TYPE ST_LaudaReadCommands_Control :
STRUCT
	SetpointOffset	: STRING := 'IN_PAR_14_';
	ControlVariable	: STRING := 'IN_MODE_01';
	OffsetSource	: STRING := 'IN_MODE_04';
END_STRUCT
END_TYPE

(* stored: Version 1.1.0.1, ProductVersion 3.1.4024.13
   DUT ST_LaudaReadCommands_Control: Id {213fd9b3-a092-4811-9e98-551440647f03} *)
